// TwinCAT 3 PLC project PLC
// ProgramVersion: 3.1.4024.0
// libraries:
//   Tc2_Standard, * (Beckhoff Automation GmbH)
//   Tc2_System, * (Beckhoff Automation GmbH)
//   Tc3_Module, * (Beckhoff Automation GmbH)
//   VisuSymbols,3.5.10.0,System
// project tree:
//   / GlobalTextList.TcGTLO, PlcTask.TcTTO, TextList.TcTLO, Visualization Manager.TcVMO (not stored), Visualization.TcVIS
//   GVLs/ GVL.TcGVL
//   POUs/ MAIN.TcPOU, Simulation01.TcPOU, Simulation02.TcPOU, TabletFillingControl02.TcPOU, TabletFillingControl01.TcPOU

CONFIGURATION PLC
    RESOURCE PLC ON TwinCAT3
        TASK PlcTask(INTERVAL := T#50000us, PRIORITY := 20);
        PROGRAM MAIN WITH PlcTask : MAIN;
    END_RESOURCE
END_CONFIGURATION

// ---- GVLs/GVL.TcGVL
{attribute 'qualified_only'}
VAR_GLOBAL
	StartPb01				:	BOOL;
	FillingPosition01		:	BOOL;
	Select3Tablet			:	BOOL;
	Select5Tablet			:	BOOL;
	Select7Tablet			:	BOOL;
	LightBarrier01			:	BOOL;
	
	MotorRunning01			:	BOOL;
	ValveOpened01			:	BOOL;
	Tablet3Selected01		:	BOOL;
	Tablet5Selected01		:	BOOL;
	Tablet7Selected01		:	BOOL;
	
	
	StartPb02				:	BOOL;
	FillingPosition02		:	BOOL;
	LightBarrier02			:	BOOL;
	
	MotorRunning02			:	BOOL;
	ValveOpened02			:	BOOL;
	TabletsSelected02		:	UINT;
	TabletsInTube02			: 	UINT;
END_VAR

// ---- POUs/MAIN.TcPOU
PROGRAM MAIN
VAR
	TabletFillingControl01	: 	TabletFillingControl01;
	TabletFillingControl02	: 	TabletFillingControl02;
END_VAR

IF FALSE THEN Simulation01(); END_IF
Simulation02();
TabletFillingControl01(
    MachineStart := GVL.StartPb01,
    FillingPosition := GVL.FillingPosition01,
    SelectTablet3 := GVL.Select3Tablet,
    SelectTablet5 := GVL.Select5Tablet,
    SelectTablet7 := GVL.Select7Tablet,
    LightBarrier := GVL.LightBarrier01);
GVL.MotorRunning01 := TabletFillingControl01.BeltMotorCmdOn;
GVL.ValveOpened01 := TabletFillingControl01.ValveCmdOpen;
GVL.Tablet3Selected01 := TabletFillingControl01.LampTablet3;
GVL.Tablet5Selected01 := TabletFillingControl01.LampTablet5;
GVL.Tablet7Selected01 := TabletFillingControl01.LampTablet7;
TabletFillingControl02(
    MachineStart := GVL.StartPb02,
    FillingPosition := GVL.FillingPosition02,
    TabletsInTube := GVL.TabletsInTube02,
    LightBarrier := GVL.LightBarrier02);
GVL.MotorRunning02 := TabletFillingControl02.BeltMotorCmdOn;
GVL.ValveOpened02 := TabletFillingControl02.ValveCmdOpen;
GVL.TabletsSelected02 := TabletFillingControl02.TabletsSelected;

END_PROGRAM

// ---- POUs/TabletFillingControl01.TcPOU
FUNCTION_BLOCK TabletFillingControl01
VAR_INPUT
	MachineStart				:	BOOL;		// True=Machine On
	FillingPosition				:	BOOL;
	SelectTablet3				:	BOOL;		// amount (3) of tablet in tube selected 
	SelectTablet5				:	BOOL;		// amount (5) of tablet in tube selected 
	SelectTablet7				:	BOOL;		// amount (7) of tablet in tube selected 
	LightBarrier				:	BOOL;		// False = free (no tablet present)
END_VAR
VAR_OUTPUT
	BeltMotorCmdOn				:	BOOL;
	ValveCmdOpen				:	BOOL;
	LampTablet3					:	BOOL;		// True = 3 tablet in tube selected
	LampTablet5					:	BOOL;		// True = 5 tablet in tube selected
	LampTablet7					:	BOOL;		// True = 7 tablet in tube selected
END_VAR
VAR
	CountTablet3				:	CTD;		// down counter for three tablets
	CountTablet5				:	CTD;		// down counter for five tablets
	CountTablet7				:	CTD;		// down counter for seven tablets
	
	Tablet3Selected				: BOOL;
	Tablet5Selected				: BOOL;
	Tablet7Selected				: BOOL;
	FirstScan					: BOOL;
	OneShot						: BOOL;			// one shot pulse after power restart		
	srTablet3Selected			: SR;
	srTablet5Selected			: SR;
	srTablet7Selected			: SR;
	
	WAIT: SR;
	SWITCHED_ON: SR;
	WAIT_FOR_FILL_POS: SR;
	FILL_POS_REACHED: SR;
	LOAD_CTR_3_TABLETS: SR;
	LOAD_CTR_5_TABLETS: SR;
	LOAD_CTR_7_TABLETS: SR;
	
	rtCount3Tablets: R_TRIG;
	rtCount5Tablets: R_TRIG;
	rtCount7Tablets: R_TRIG;
	tonCount3Tablet: TON;
	tonCount5Tablet: TON;
	tonCount7Tablet: TON;
END_VAR
VAR // added by the converter: edge detectors and wires of the graphical bodies
    _w1 : BOOL;
END_VAR

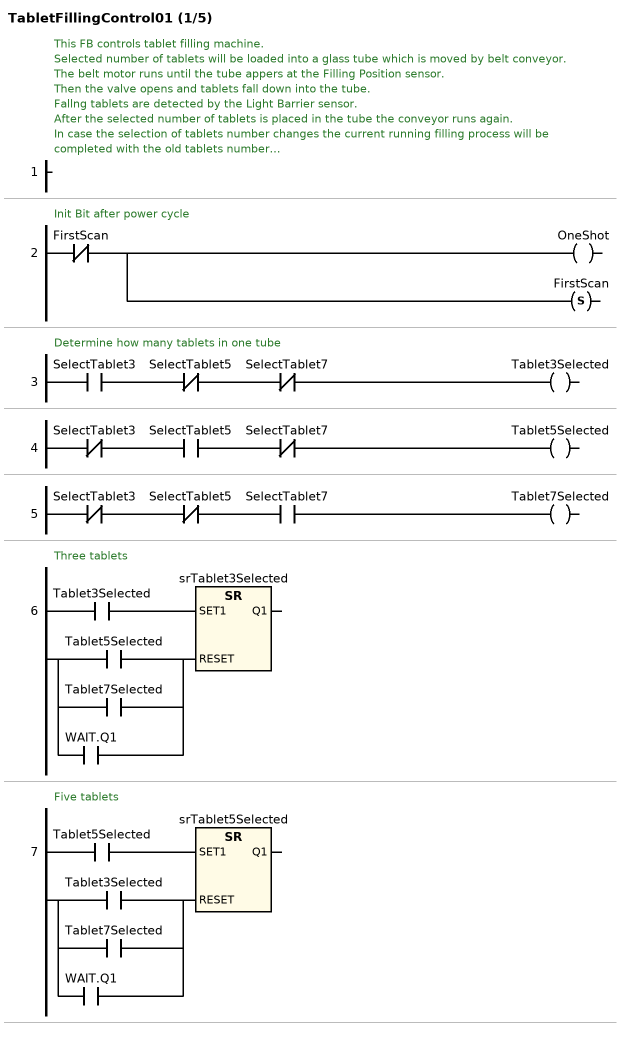
// NETWORK 1
// This FB controls tablet filling machine.
// Selected number of tablets will be loaded into a glass tube which is moved by belt conveyor.
// The belt motor runs until the tube appers at the Filling Position sensor.
// Then the valve opens and tablets fall down into the tube.
// Fallng tablets are detected by the Light Barrier sensor.
// After the selected number of tablets is placed in the tube the conveyor runs again.
// In case the selection of tablets number changes the current running filling process will be completed with the old tablets number.
// This is Version 01 of the program - only three fixed number (3,5,7) of tablets can be chosen by boolean input.

// NETWORK 2
// Init Bit after power cycle
_w1 := NOT FirstScan;
OneShot := _w1;
FirstScan S= _w1;

// NETWORK 3
// Determine how many tablets in one tube
Tablet3Selected := SelectTablet3 AND NOT SelectTablet5 AND NOT SelectTablet7;

// NETWORK 4
Tablet5Selected := NOT SelectTablet3 AND SelectTablet5 AND NOT SelectTablet7;

// NETWORK 5
Tablet7Selected := NOT SelectTablet3 AND NOT SelectTablet5 AND SelectTablet7;

// NETWORK 6
// Three tablets
srTablet3Selected(SET1 := Tablet3Selected, RESET := Tablet5Selected OR Tablet7Selected OR WAIT.Q1); // SR

// NETWORK 7
// Five tablets
srTablet5Selected(SET1 := Tablet5Selected, RESET := Tablet3Selected OR Tablet7Selected OR WAIT.Q1); // SR

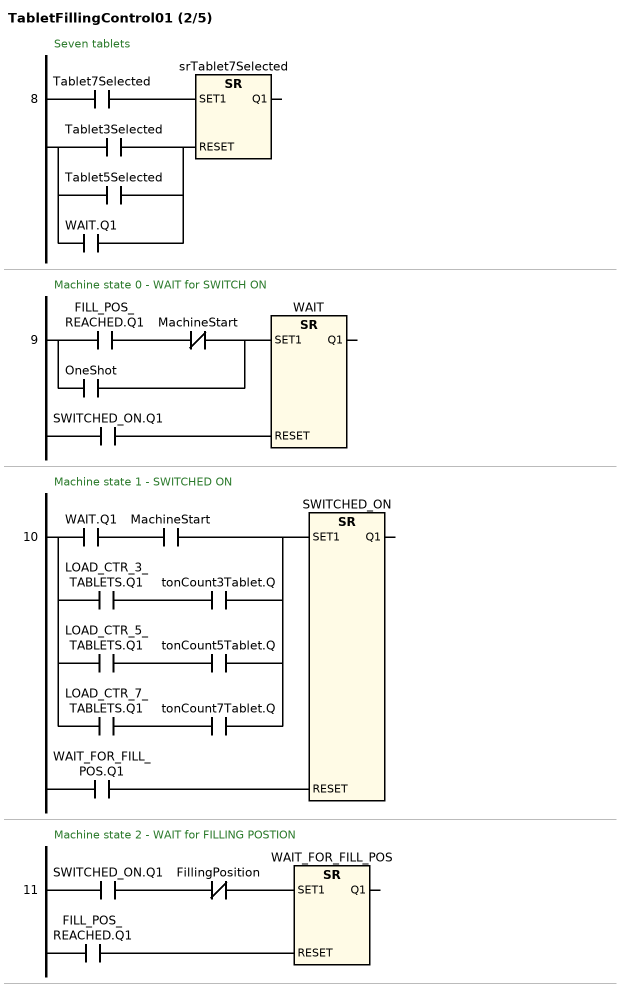
// NETWORK 8
// Seven tablets
srTablet7Selected(SET1 := Tablet7Selected, RESET := Tablet3Selected OR Tablet5Selected OR WAIT.Q1); // SR

// NETWORK 9
// Machine state 0 - WAIT for SWITCH ON
WAIT(SET1 := FILL_POS_REACHED.Q1 AND NOT MachineStart OR OneShot, RESET := SWITCHED_ON.Q1); // SR

// NETWORK 10
// Machine state 1 - SWITCHED ON
SWITCHED_ON(SET1 := WAIT.Q1 AND MachineStart OR LOAD_CTR_3_TABLETS.Q1 AND tonCount3Tablet.Q OR LOAD_CTR_5_TABLETS.Q1 AND tonCount5Tablet.Q OR LOAD_CTR_7_TABLETS.Q1 AND tonCount7Tablet.Q, RESET := WAIT_FOR_FILL_POS.Q1); // SR

// NETWORK 11
// Machine state 2 - WAIT for FILLING POSTION
WAIT_FOR_FILL_POS(SET1 := SWITCHED_ON.Q1 AND NOT FillingPosition, RESET := FILL_POS_REACHED.Q1); // SR

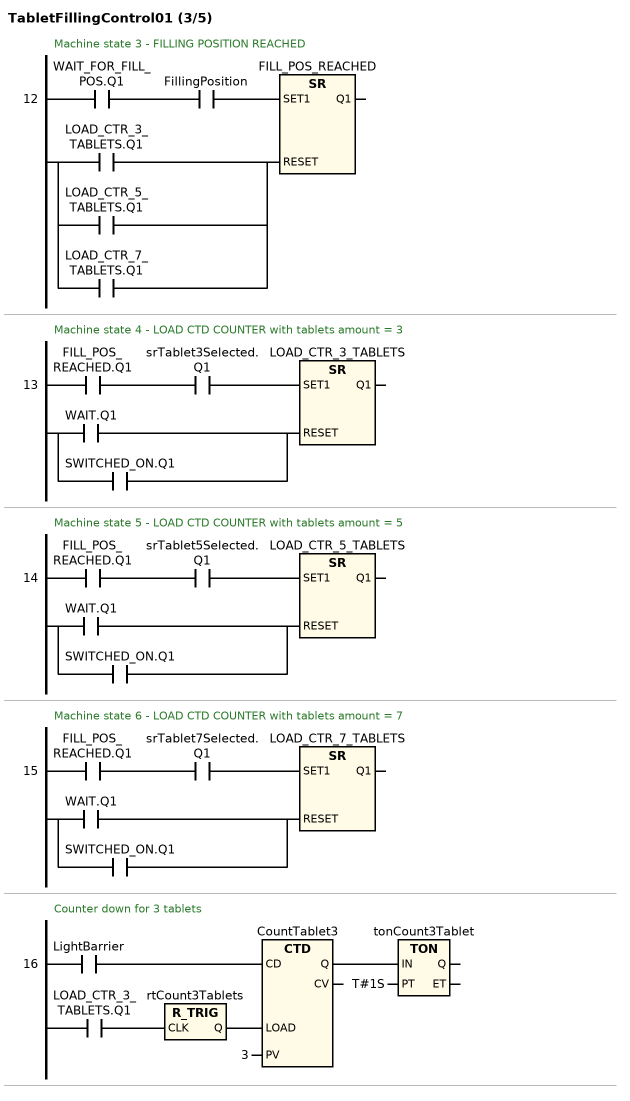
// NETWORK 12
// Machine state 3 - FILLING POSITION REACHED
FILL_POS_REACHED(SET1 := WAIT_FOR_FILL_POS.Q1 AND FillingPosition, RESET := LOAD_CTR_3_TABLETS.Q1 OR LOAD_CTR_5_TABLETS.Q1 OR LOAD_CTR_7_TABLETS.Q1); // SR

// NETWORK 13
// Machine state 4 - LOAD CTD COUNTER with tablets amount = 3
LOAD_CTR_3_TABLETS(SET1 := FILL_POS_REACHED.Q1 AND srTablet3Selected.Q1, RESET := WAIT.Q1 OR SWITCHED_ON.Q1); // SR

// NETWORK 14
// Machine state 5 - LOAD CTD COUNTER with tablets amount = 5
LOAD_CTR_5_TABLETS(SET1 := FILL_POS_REACHED.Q1 AND srTablet5Selected.Q1, RESET := WAIT.Q1 OR SWITCHED_ON.Q1); // SR

// NETWORK 15
// Machine state 6 - LOAD CTD COUNTER with tablets amount = 7
LOAD_CTR_7_TABLETS(SET1 := FILL_POS_REACHED.Q1 AND srTablet7Selected.Q1, RESET := WAIT.Q1 OR SWITCHED_ON.Q1); // SR

// NETWORK 16
// Counter down for 3 tablets
rtCount3Tablets(CLK := LOAD_CTR_3_TABLETS.Q1); // R_TRIG
CountTablet3(CD := LightBarrier, LOAD := rtCount3Tablets.Q, PV := 3); // CTD
tonCount3Tablet(IN := CountTablet3.Q, PT := T#1S); // TON

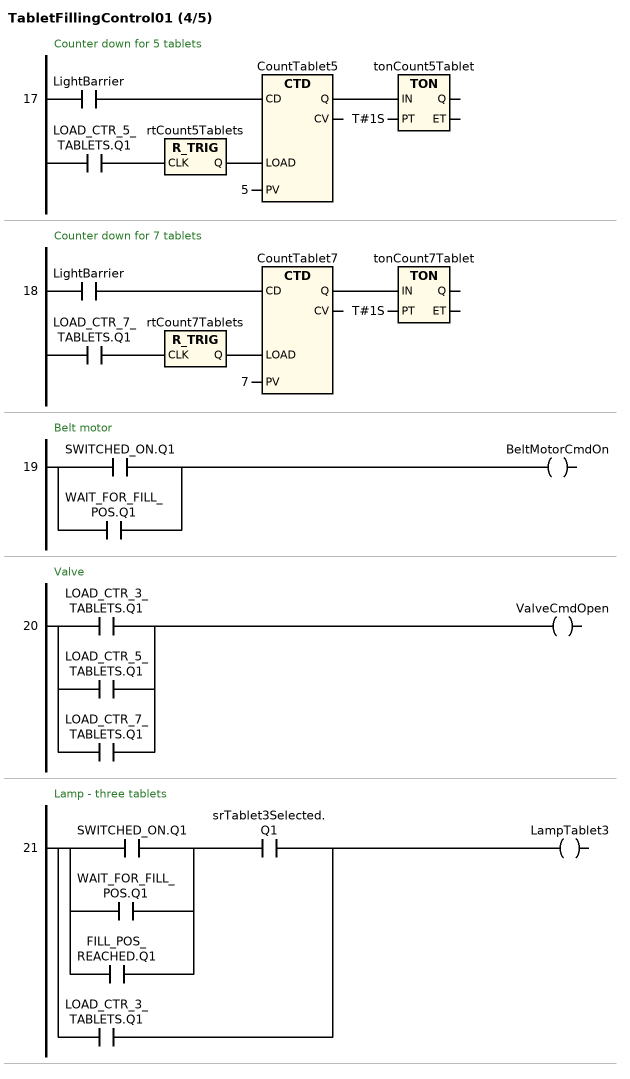
// NETWORK 17
// Counter down for 5 tablets
rtCount5Tablets(CLK := LOAD_CTR_5_TABLETS.Q1); // R_TRIG
CountTablet5(CD := LightBarrier, LOAD := rtCount5Tablets.Q, PV := 5); // CTD
tonCount5Tablet(IN := CountTablet5.Q, PT := T#1S); // TON

// NETWORK 18
// Counter down for 7 tablets
rtCount7Tablets(CLK := LOAD_CTR_7_TABLETS.Q1); // R_TRIG
CountTablet7(CD := LightBarrier, LOAD := rtCount7Tablets.Q, PV := 7); // CTD
tonCount7Tablet(IN := CountTablet7.Q, PT := T#1S); // TON

// NETWORK 19
// Belt motor
BeltMotorCmdOn := SWITCHED_ON.Q1 OR WAIT_FOR_FILL_POS.Q1;

// NETWORK 20
// Valve
ValveCmdOpen := LOAD_CTR_3_TABLETS.Q1 OR LOAD_CTR_5_TABLETS.Q1 OR LOAD_CTR_7_TABLETS.Q1;

// NETWORK 21
// Lamp - three tablets
LampTablet3 := (SWITCHED_ON.Q1 OR WAIT_FOR_FILL_POS.Q1 OR FILL_POS_REACHED.Q1) AND srTablet3Selected.Q1 OR LOAD_CTR_3_TABLETS.Q1;

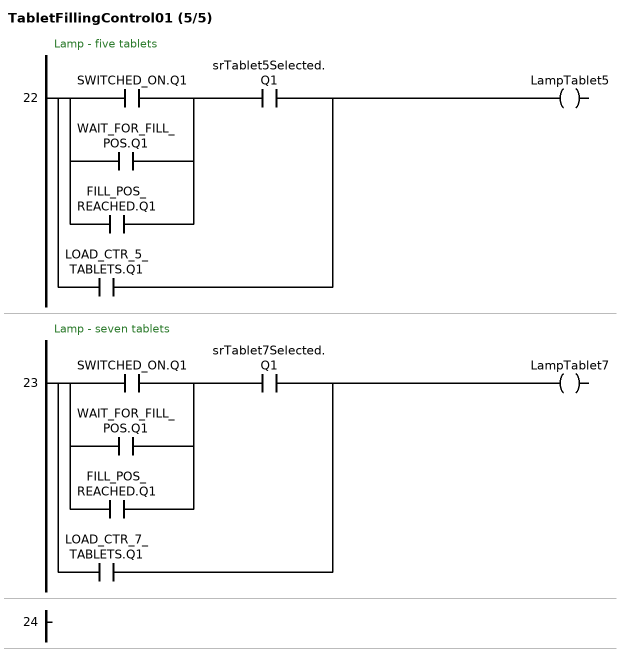
// NETWORK 22
// Lamp - five tablets
LampTablet5 := (SWITCHED_ON.Q1 OR WAIT_FOR_FILL_POS.Q1 OR FILL_POS_REACHED.Q1) AND srTablet5Selected.Q1 OR LOAD_CTR_5_TABLETS.Q1;

// NETWORK 23
// Lamp - seven tablets
LampTablet7 := (SWITCHED_ON.Q1 OR WAIT_FOR_FILL_POS.Q1 OR FILL_POS_REACHED.Q1) AND srTablet7Selected.Q1 OR LOAD_CTR_7_TABLETS.Q1;

// NETWORK 24

END_FUNCTION_BLOCK

// ---- POUs/TabletFillingControl02.TcPOU
FUNCTION_BLOCK TabletFillingControl02
VAR_INPUT
	MachineStart				:	BOOL;		// True=Machine On
	FillingPosition				:	BOOL;		// Tube in loading position
	TabletsInTube				:	UINT;		// Number of tablets which should be loaded into one tube
	LightBarrier				:	BOOL;		// False=free (no tablet present), True=tablet present
END_VAR
VAR_OUTPUT
	BeltMotorCmdOn				:	BOOL;		// Belt motor command ON
	ValveCmdOpen				:	BOOL;		// Valve command OPEN
	TabletsSelected				:	UINT;		// Number of tablet selected to be loaded into one tube
END_VAR
VAR
	ctdTablets					: CTD;		// down counter for three tablets
	
	FirstScan					: BOOL;
	OneShot						: BOOL;		// one shot pulse after power restart		
	srTabletNumberSelected		: SR;		// Number of tablets properly selected (>0)

	WAIT						: BOOL;		// Machine state 'Wait'
	SWITCHED_ON					: BOOL;		// Machine state 'Switched on'
	WAIT_FOR_FILL_POS			: BOOL;		// Machine state 'Waiting for filling position'
	FILL_POS_REACHED			: BOOL;		// Machine state 'Filling position reached'
	LOAD_CTR_TABLETS			: BOOL;		// Machine state 'Load counter with tablets number'

	
	rtTabletCntrLoaded			: R_TRIG;	// Tablet counter loaded with number of tablet
	tonCountTablet				: TON;		// delay after last tablet detected to allow proper positioning in the tube
END_VAR
VAR // added by the converter: edge detectors and wires of the graphical bodies
    _w1 : BOOL;
END_VAR

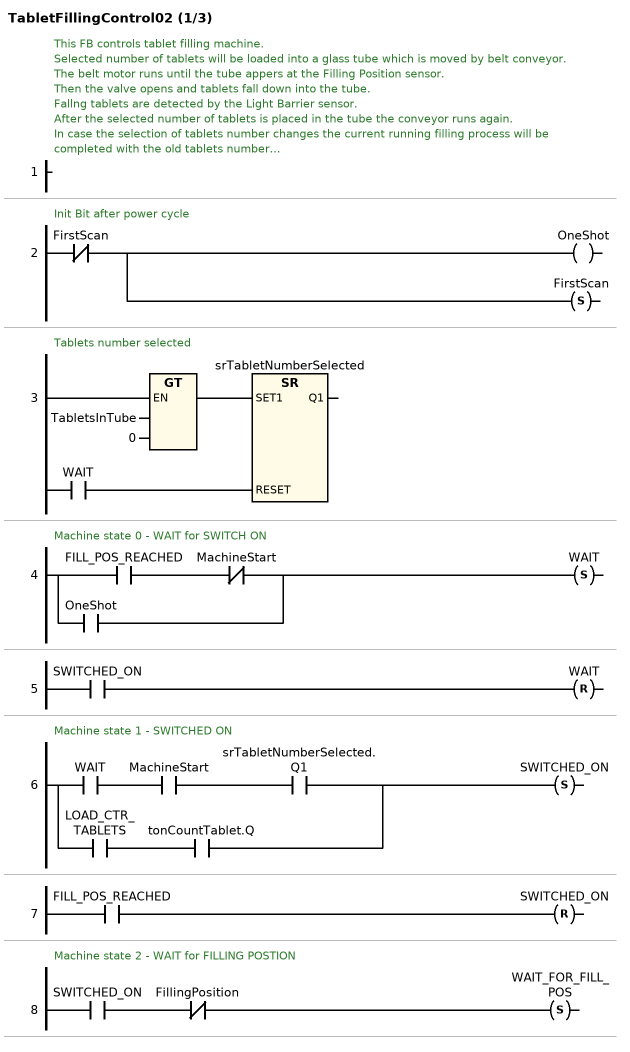
// NETWORK 1
// This FB controls tablet filling machine.
// Selected number of tablets will be loaded into a glass tube which is moved by belt conveyor.
// The belt motor runs until the tube appers at the Filling Position sensor.
// Then the valve opens and tablets fall down into the tube.
// Fallng tablets are detected by the Light Barrier sensor.
// After the selected number of tablets is placed in the tube the conveyor runs again.
// In case the selection of tablets number changes the current running filling process will be completed with the old tablets number.
// This is Version 02 of the program - any number number of tablets can be chosen by 'TabletsInTube' variable

// NETWORK 2
// Init Bit after power cycle
_w1 := NOT FirstScan;
OneShot := _w1;
FirstScan S= _w1;

// NETWORK 3
// Tablets number selected
srTabletNumberSelected(SET1 := TabletsInTube > 0, RESET := WAIT); // SR

// NETWORK 4
// Machine state 0 - WAIT for SWITCH ON
WAIT S= FILL_POS_REACHED AND NOT MachineStart OR OneShot;

// NETWORK 5
WAIT R= SWITCHED_ON;

// NETWORK 6
// Machine state 1 - SWITCHED ON
SWITCHED_ON S= WAIT AND MachineStart AND srTabletNumberSelected.Q1 OR LOAD_CTR_TABLETS AND tonCountTablet.Q;

// NETWORK 7
SWITCHED_ON R= FILL_POS_REACHED;

// NETWORK 8
// Machine state 2 - WAIT for FILLING POSTION
WAIT_FOR_FILL_POS S= SWITCHED_ON AND NOT FillingPosition;

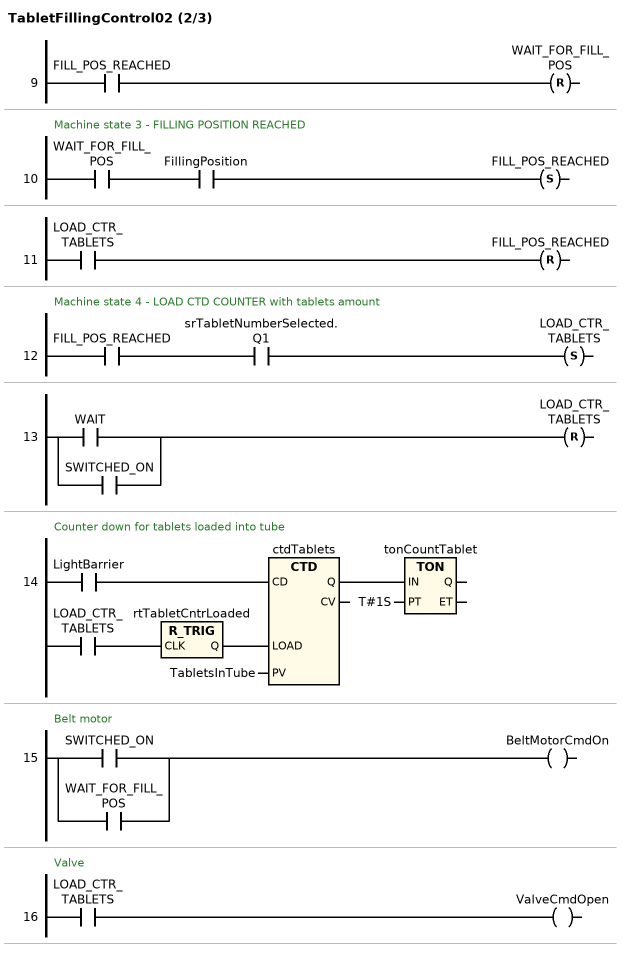
// NETWORK 9
WAIT_FOR_FILL_POS R= FILL_POS_REACHED;

// NETWORK 10
// Machine state 3 - FILLING POSITION REACHED
FILL_POS_REACHED S= WAIT_FOR_FILL_POS AND FillingPosition;

// NETWORK 11
FILL_POS_REACHED R= LOAD_CTR_TABLETS;

// NETWORK 12
// Machine state 4 - LOAD CTD COUNTER with tablets amount
LOAD_CTR_TABLETS S= FILL_POS_REACHED AND srTabletNumberSelected.Q1;

// NETWORK 13
LOAD_CTR_TABLETS R= WAIT OR SWITCHED_ON;

// NETWORK 14
// Counter down for tablets loaded into tube
rtTabletCntrLoaded(CLK := LOAD_CTR_TABLETS); // R_TRIG
ctdTablets(CD := LightBarrier, LOAD := rtTabletCntrLoaded.Q, PV := TabletsInTube); // CTD
tonCountTablet(IN := ctdTablets.Q, PT := T#1S); // TON

// NETWORK 15
// Belt motor
BeltMotorCmdOn := SWITCHED_ON OR WAIT_FOR_FILL_POS;

// NETWORK 16
// Valve
ValveCmdOpen := LOAD_CTR_TABLETS;

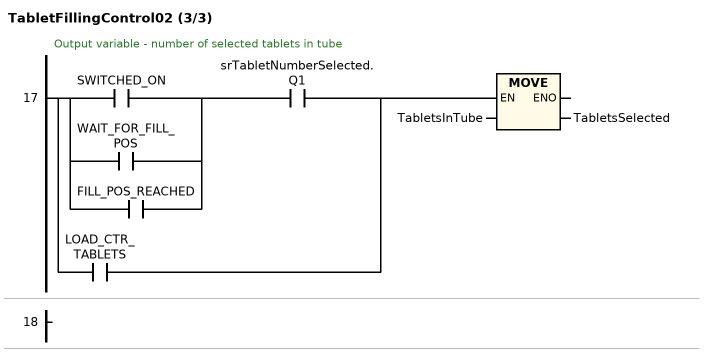
// NETWORK 17
// Output variable - number of selected tablets in tube
IF (SWITCHED_ON OR WAIT_FOR_FILL_POS OR FILL_POS_REACHED) AND srTabletNumberSelected.Q1 OR LOAD_CTR_TABLETS THEN
    TabletsSelected := TabletsInTube;
END_IF

// NETWORK 18

END_FUNCTION_BLOCK

// ---- POUs/Simulation01.TcPOU
PROGRAM Simulation01
VAR
	TubePosition					:	ARRAY[1..3] OF UINT :=[0,0,0];
	OffsetForNextTube				:	UINT := 90;				
	Idx								:	UINT;
	TubePosStep						:	UINT := 1;
	Tube02Active					:	BOOL;
	Tube03Active					:	BOOL;
	FillingPos						:	UINT := 275;
	ValvePosition					:	UINT;
	NewTubeFilling					:	BOOL;
	TabletPositionVert				: 	UINT;
	TabletPositionHorizn			: 	UINT;
	TabletNumberInTube				:	UINT;
	TabletNumberLoaded				:	UINT;
	
	VisuTabletsInTube				:	UINT;
END_VAR

IF VisuTabletsInTube = 0 THEN
	GVL.Select3Tablet := TRUE;
	GVL.Select5Tablet := FALSE;
	GVL.Select7Tablet := FALSE;
ELSIF VisuTabletsInTube = 1 THEN
	GVL.Select3Tablet := FALSE;
	GVL.Select5Tablet := TRUE;
	GVL.Select7Tablet := FALSE;
ELSIF VisuTabletsInTube = 2 THEN
	GVL.Select3Tablet := FALSE;
	GVL.Select5Tablet := FALSE;
	GVL.Select7Tablet := TRUE;
END_IF


IF GVL.MotorRunning01 THEN
	
	(* tube motion simulation *)
	TubePosition[1] := SEL(TubePosition[1] <= 330, 0, TubePosition[1] + TubePosStep);
	IF TubePosition[1] > OffsetForNextTube THEN
		Tube02Active := TRUE;
	END_IF
	
	IF Tube02Active THEN
		TubePosition[2] := SEL(TubePosition[2] <= 330, 0, TubePosition[2] + TubePosStep);
	END_IF
	Tube02Active := TubePosition[2] >0 AND TubePosition[2] <=330;
	
	IF TubePosition[2] > OffsetForNextTube THEN
		Tube03Active := TRUE;
	END_IF
	
	IF Tube03Active THEN
		TubePosition[3] := SEL(TubePosition[3] <= 330, 0, TubePosition[3] + TubePosStep);
	END_IF
	Tube03Active := TubePosition[3] >0 AND TubePosition[3] <=330;
	
	// check if any tube at the filling position
	FOR Idx:= 1 TO 3 DO
		IF ABS(FillingPos - TubePosition[Idx]) < 2  THEN
			GVL.FillingPosition01 := TRUE;
			// some tube at the filling position, not needed to test anothers 
			EXIT;
		ELSE
			GVL.FillingPosition01 := FALSE;
		END_IF
	END_FOR
	
	// tube loaded with selected number of tablets, move tablets together with tube 
	IF TabletNumberLoaded = TabletNumberInTube THEN
		TabletPositionHorizn := TabletPositionHorizn + TubePosStep;
	END_IF
	
	// check if any tablets with tube on the end of belt conveyor
	FOR Idx:= 1 TO 3 DO
		IF ABS(330 - TubePosition[Idx]) < 2 THEN
			TabletNumberLoaded := 0;
			TabletPositionHorizn := 0;
		END_IF
	END_FOR
	
	
	
END_IF



// valve simulation
IF GVL.ValveOpened01 THEN
	ValvePosition := 24;
	NewTubeFilling := TRUE;
ELSE
	ValvePosition := 0;
	NewTubeFilling := FALSE;
END_IF

// falling tablet simulation
IF GVL.Select3Tablet THEN 
	TabletNumberInTube := 3;
ELSIF GVL.Select5Tablet THEN 
	TabletNumberInTube := 5;
ELSIF GVL.Select7Tablet THEN 
	TabletNumberInTube := 7; 
END_IF;


IF NewTubeFilling AND TabletNumberLoaded < TabletNumberInTube THEN
	TabletPositionVert := TabletPositionVert + 2;
	// tablet position in tube
	IF TabletPositionVert >= 69 THEN
		TabletNumberLoaded := TabletNumberLoaded+1;
		TabletPositionVert := 0;
	END_IF
END_IF


// Light barrier simulation
GVL.LightBarrier01 := TabletPositionVert > 36 AND TabletPositionVert < 46;

END_PROGRAM

// ---- POUs/Simulation02.TcPOU
PROGRAM Simulation02
VAR
	TubePosition					:	ARRAY[1..3] OF UINT :=[0,0,0];
	OffsetForNextTube				:	UINT := 90;				
	Idx								:	UINT;
	TubePosStep						:	UINT := 1;
	Tube02Active					:	BOOL;
	Tube03Active					:	BOOL;
	FillingPos						:	UINT := 275;
	ValvePosition					:	UINT;
	NewTubeFilling					:	BOOL;
	TabletPositionVert				: 	UINT;
	TabletPositionHorizn			: 	UINT;
	TabletNumberInTube				:	UINT;
	TabletNumberLoaded				:	UINT;
	
	VisuTabletsInTube				:	UINT;
END_VAR

GVL.TabletsInTube02 := VisuTabletsInTube;

IF GVL.MotorRunning02 THEN
	
	(* tube motion simulation *)
	TubePosition[1] := SEL(TubePosition[1] <= 330, 0, TubePosition[1] + TubePosStep);
	IF TubePosition[1] > OffsetForNextTube THEN
		Tube02Active := TRUE;
	END_IF
	
	IF Tube02Active THEN
		TubePosition[2] := SEL(TubePosition[2] <= 330, 0, TubePosition[2] + TubePosStep);
	END_IF
	Tube02Active := TubePosition[2] >0 AND TubePosition[2] <=330;
	
	IF TubePosition[2] > OffsetForNextTube THEN
		Tube03Active := TRUE;
	END_IF
	
	IF Tube03Active THEN
		TubePosition[3] := SEL(TubePosition[3] <= 330, 0, TubePosition[3] + TubePosStep);
	END_IF
	Tube03Active := TubePosition[3] >0 AND TubePosition[3] <=330;
	
	// check if any tube at the filling position
	FOR Idx:= 1 TO 3 DO
		IF ABS(FillingPos - TubePosition[Idx]) < 2  THEN
			GVL.FillingPosition02 := TRUE;
			// some tube at the filling position, not needed to test anothers 
			EXIT;
		ELSE
			GVL.FillingPosition02 := FALSE;
		END_IF
	END_FOR
	
	// tube loaded with selected number of tablets, move tablets together with tube 
	IF TabletNumberLoaded = TabletNumberInTube THEN
		TabletPositionHorizn := TabletPositionHorizn + TubePosStep;
	END_IF
	
	// check if any tablets with tube on the end of belt conveyor
	FOR Idx:= 1 TO 3 DO
		IF ABS(330 - TubePosition[Idx]) < 2 THEN
			TabletNumberLoaded := 0;
			TabletPositionHorizn := 0;
		END_IF
	END_FOR
	
	
	
END_IF



// valve simulation
IF GVL.ValveOpened02 THEN
	ValvePosition := 24;
	NewTubeFilling := TRUE;
ELSE
	ValvePosition := 0;
	NewTubeFilling := FALSE;
END_IF


// falling tablet simulation
TabletNumberInTube := GVL.TabletsInTube02;


IF NewTubeFilling AND TabletNumberLoaded < TabletNumberInTube THEN
	TabletPositionVert := TabletPositionVert + 2;
	// tablet position in tube
	IF TabletPositionVert >= 69 THEN
		TabletNumberLoaded := TabletNumberLoaded+1;
		TabletPositionVert := 0;
	END_IF
END_IF


// Light barrier simulation
GVL.LightBarrier02 := TabletPositionVert > 36 AND TabletPositionVert < 46;

END_PROGRAM

// ---- GlobalTextList.TcGTLO
TEXTLIST GlobalTextList
  542 = 'Change Tray'
  369 = 'Filling Position \nSensor'
  941 = 'Filling Position Sensor'
  242 = 'FillingPositionBarrier'
  800 = 'Five tablets in tube'
  722 = 'Light Barrier'
  329 = 'Motor'
  959 = 'Please Change the Tray'
  663 = 'Product amount: \n%s'
  814 = 'RUN'
  60 = 'Select number of \ntablets in tube: \n%s'
  105 = 'Select number of tablets in tube: \n%s'
  25 = 'Seven tablets in tube'
  183 = 'START'
  872 = 'STOP'
  349 = 'Tablets'
  323 = 'Tablets in tube selected: \n%s'
  240 = 'Three tablets in tube'
  513 = 'Tube'
  338 = 'Valve'
END_TEXTLIST

// ---- TextList.TcTLO
TEXTLIST TextList
  0 = '0'
  1 = '1'
  2 = '3'
  4 = '5'
  6 = '6'
  7 = '7'
  8 = '8'
  9 = '9'
  10 = '10'
   = ''
END_TEXTLIST

// ---- Visualization.TcVIS
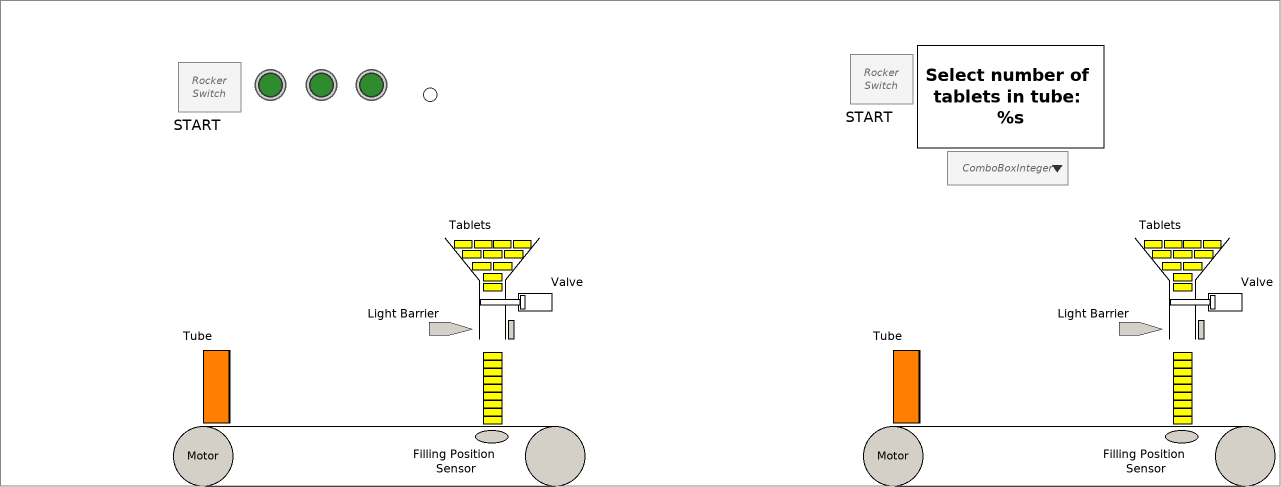
VISUALIZATION Visualization  // 1281x487
    Rectangle (518,293 34x18)
    Rectangle (917,45 187x103), "Select number of tablets in tube: %s", text variable: GVL.TabletsSelected02
    Ellipse (173,426 60x60), "Motor", colour toggle: GVL.MotorRunning01
    Ellipse (525,426 60x60), colour toggle: GVL.MotorRunning01
    Line (205,486) (555,486), colour toggle: GVL.MotorRunning01
    Line (202,426) (555,426), colour toggle: GVL.MotorRunning01
    Label (408,443 96x37), "Filling Position Sensor"
    Rectangle (204,350 26x73)
        p3560616238: Simulation01.TubePosition[1]
    Line (479,280) (479,339)
    Line (505,280) (505,339)
    Line (539,238) (505,280)
    Group (480,295 45x14)
        p3560616238: Simulation01.ValvePosition
        Rectangle (0,4 40x6)
        Rectangle (40,0 5x14)
    Line (479,280) (445,238)
    RoundedRectangle (483,283 19x8)
        p2738717112: Simulation01.TabletPositionVert
    RoundedRectangle (454,240 18x8)
    RoundedRectangle (462,250 19x8)
    RoundedRectangle (472,262 19x8)
    RoundedRectangle (483,273 19x8)
    RoundedRectangle (483,250 19x8)
    RoundedRectangle (493,262 19x8)
    RoundedRectangle (504,250 19x8)
    RoundedRectangle (493,240 18x8)
    RoundedRectangle (474,240 18x8)
    RoundedRectangle (513,240 18x8)
    Ellipse (475,430 33x13), colour toggle: GVL.FillingPosition01
    Label (543,271 48x22), "Valve"
    Label (446,214 48x22), "Tablets"
    Label (171,325 53x22), "Tube"
    Polygon (429,322) (449,322) (472,329) (449,335) (429,335), colour toggle: GVL.LightBarrier01
    Label (355,301 96x25), "Light Barrier"
    Rectangle (508,320 6x19)
    Rectangle (203,350 26x73), invisible if: NOT Simulation01.Tube02Active
        p3560616238: Simulation01.TubePosition[2]
    Rectangle (203,350 26x73), invisible if: NOT Simulation01.Tube03Active
        p3560616238: Simulation01.TubePosition[3]
    RoundedRectangle (483,416 19x8), invisible if: Simulation01.TabletNumberLoaded = 0
        p3560616238: Simulation01.TabletPositionHorizn
    RoundedRectangle (483,408 19x8), invisible if: Simulation01.TabletNumberLoaded < 2
        p3560616238: Simulation01.TabletPositionHorizn
    RoundedRectangle (483,400 19x8), invisible if: Simulation01.TabletNumberLoaded < 3
        p3560616238: Simulation01.TabletPositionHorizn
    RoundedRectangle (483,392 19x8), invisible if: Simulation01.TabletNumberLoaded < 4
        p3560616238: Simulation01.TabletPositionHorizn
    RoundedRectangle (483,384 19x8), invisible if: Simulation01.TabletNumberLoaded < 5
        p3560616238: Simulation01.TabletPositionHorizn
    RoundedRectangle (483,376 19x8), invisible if: Simulation01.TabletNumberLoaded < 6
        p3560616238: Simulation01.TabletPositionHorizn
    RoundedRectangle (483,368 19x8), invisible if: Simulation01.TabletNumberLoaded < 7
        p3560616238: Simulation01.TabletPositionHorizn
    RoundedRectangle (483,360 19x8), invisible if: Simulation01.TabletNumberLoaded < 8
        p3560616238: Simulation01.TabletPositionHorizn
    RoundedRectangle (483,352 19x8), invisible if: Simulation01.TabletNumberLoaded < 9
        p3560616238: Simulation01.TabletPositionHorizn
    Lamp1 (252,64 37x42), variable: GVL.Tablet3Selected01, style: Lamp-Lamp1-Green
    RockerSwitch (178,62 63x50), variable: GVL.StartPb01, behaviour: TOGGLE, style: Switch-RockerSwitch-Blue
    Label (156,114 82x22), "START"
    Lamp1 (303,64 37x42), variable: GVL.Tablet5Selected01, style: Lamp-Lamp1-Green
    Lamp1 (353,64 37x42), variable: GVL.Tablet7Selected01, style: Lamp-Lamp1-Green
    RadioButton (421,41 192x107), variable: Simulation01.VisuTabletsInTube
        Areas[0]: Text=Three tablets in tube
        Areas[1]: Text=Five tablets in tube
        Areas[2]: Text=Seven tablets in tube
    ComboBoxInteger (947,151 121x34), variable: Simulation02.VisuTabletsInTube
    RockerSwitch (850,54 63x50), variable: GVL.StartPb02, behaviour: TOGGLE, style: Switch-RockerSwitch-Blue
    Label (828,106 82x22), "START"
    Rectangle (1208,293 34x18)
    Ellipse (863,426 60x60), "Motor", colour toggle: GVL.MotorRunning02
    Ellipse (1215,426 60x60), colour toggle: GVL.MotorRunning02
    Line (895,486) (1245,486), colour toggle: GVL.MotorRunning02
    Line (892,426) (1245,426), colour toggle: GVL.MotorRunning02
    Label (1098,443 96x37), "Filling Position Sensor"
    Rectangle (894,350 26x73)
        p3560616238: Simulation02.TubePosition[1]
    Line (1169,280) (1169,339)
    Line (1195,280) (1195,339)
    Line (1229,238) (1195,280)
    Group (1170,295 45x14)
        p3560616238: Simulation02.ValvePosition
        Rectangle (0,4 40x6)
        Rectangle (40,0 5x14)
    Line (1169,280) (1135,238)
    RoundedRectangle (1173,283 19x8)
        p2738717112: Simulation02.TabletPositionVert
    RoundedRectangle (1144,240 18x8)
    RoundedRectangle (1152,250 19x8)
    RoundedRectangle (1162,262 19x8)
    RoundedRectangle (1173,273 19x8)
    RoundedRectangle (1173,250 19x8)
    RoundedRectangle (1183,262 19x8)
    RoundedRectangle (1194,250 19x8)
    RoundedRectangle (1183,240 18x8)
    RoundedRectangle (1164,240 18x8)
    RoundedRectangle (1203,240 18x8)
    Ellipse (1165,430 33x13), colour toggle: GVL.FillingPosition02
    Label (1233,271 48x22), "Valve"
    Label (1136,214 48x22), "Tablets"
    Label (861,325 53x22), "Tube"
    Polygon (1119,322) (1139,322) (1162,329) (1139,335) (1119,335), colour toggle: GVL.LightBarrier02
    Label (1045,301 96x25), "Light Barrier"
    Rectangle (1198,320 6x19)
    Rectangle (893,350 26x73), invisible if: NOT Simulation02.Tube02Active
        p3560616238: Simulation02.TubePosition[2]
    Rectangle (893,350 26x73), invisible if: NOT Simulation02.Tube03Active
        p3560616238: Simulation02.TubePosition[3]
    RoundedRectangle (1173,416 19x8), invisible if: Simulation02.TabletNumberLoaded = 0
        p3560616238: Simulation02.TabletPositionHorizn
    RoundedRectangle (1173,408 19x8), invisible if: Simulation02.TabletNumberLoaded < 2
        p3560616238: Simulation02.TabletPositionHorizn
    RoundedRectangle (1173,400 19x8), invisible if: Simulation02.TabletNumberLoaded < 3
        p3560616238: Simulation02.TabletPositionHorizn
    RoundedRectangle (1173,392 19x8), invisible if: Simulation02.TabletNumberLoaded < 4
        p3560616238: Simulation02.TabletPositionHorizn
    RoundedRectangle (1173,384 19x8), invisible if: Simulation02.TabletNumberLoaded < 5
        p3560616238: Simulation02.TabletPositionHorizn
    RoundedRectangle (1173,376 19x8), invisible if: Simulation02.TabletNumberLoaded < 6
        p3560616238: Simulation02.TabletPositionHorizn
    RoundedRectangle (1173,368 19x8), invisible if: Simulation02.TabletNumberLoaded < 7
        p3560616238: Simulation02.TabletPositionHorizn
    RoundedRectangle (1173,360 19x8), invisible if: Simulation02.TabletNumberLoaded < 8
        p3560616238: Simulation02.TabletPositionHorizn
    RoundedRectangle (1173,352 19x8), invisible if: Simulation02.TabletNumberLoaded < 9
        p3560616238: Simulation02.TabletPositionHorizn
END_VISUALIZATION
